FUNCTION_BLOCK STATION3
  {SET_ATTRIBUTE(OpcUa, DEVICE.SENSOR)}
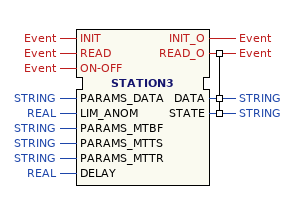
  EVENT_INPUT
    INIT;
    READ;
    ON-OFF;
  END_EVENT
  EVENT_OUTPUT
    INIT_O;
    READ_O WITH DATA, STATE;
  END_EVENT
  VAR_INPUT
    PARAMS_DATA : STRING;
    LIM_ANOM : REAL;
    PARAMS_MTBF : STRING;
    PARAMS_MTTS : STRING;
    PARAMS_MTTR : STRING;
    DELAY : REAL;
  END_VAR
  VAR_OUTPUT
    DATA : STRING;
    STATE : STRING;
  END_VAR
END_FUNCTION_BLOCK
